(* IEC 61131-3 sources: CodesysTest/alpha/export/FBs/DelayDwellFB/DelayDwellFB.pou/DwellSetting.prop, 1 file *)

(* ---- Get.pm.st ---- *)
(*#-#-#-#-#-#-#-#-#-#---Declaration---#-#-#-#-#-#-#-#-#-#-#-#-#*)

VAR
END_VAR
(*#-#-#-#-#-#-#-#-#-#---Implementation---#-#-#-#-#-#-#-#-#-#-#-#-#*)

DwellSetting := _dwellTimeInMS;
